// Mitsubishi GX Works2 project: sm샘플   PLC: Q02/Q02H

PROGRAM MAIN
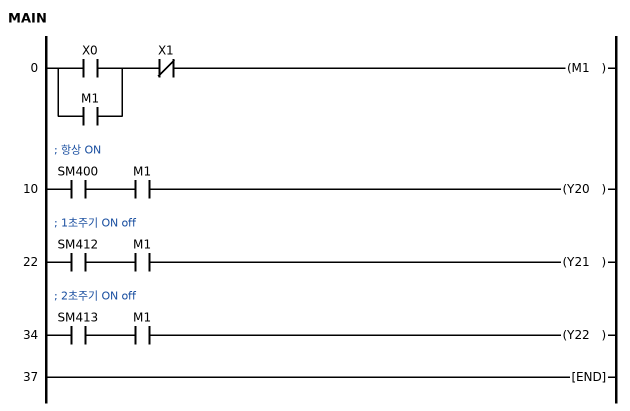
0     LD      X0
      OR      M1
      ANI     X1
      OUT     M1
; 항상 ON
10    LD      SM400
      AND     M1
      OUT     Y20
; 1초주기 ON off
22    LD      SM412
      AND     M1
      OUT     Y21
; 2초주기 ON off
34    LD      SM413
      AND     M1
      OUT     Y22
37    END
END_PROGRAM
